(* PLC project PlainProject, Unknown Unnamed 1 *)
(* stored: creationDateTime 2023-09-14T08:06:45, modificationDateTime 2023-09-14T08:09:26 *)

PROGRAM program0
  VAR
    inlet AT %MW0.0.0.20 : INT;
    outlet AT %MW0.0.0.21 : INT;
    level AT %MW0.0.1.0 : INT;
    statustank AT %MW0.0.2.0 : INT;
  END_VAR
  VAR
    pv : INT;
    sp : INT;
    state : INT;
    Setpoint : INT;
    ValveButtonBoth : BOOL;
    tankstatus : INT;
  END_VAR

            pv := level;
sp := Setpoint;
tankstatus := statustank; (* 1=OK, 2=WARNING, 3=BROKEN *)

if ValveButtonBoth then 
state := 4;
else
if pv >= 90 then
state := 1; (* 0= HOLD,  1= DUMP (to not anger management), 2= DRAIN, 3:= FILL *) 
elsif pv > sp + 3 then
state := 2;
elsif pv < sp - 3 then
state :=3;
else
state :=0;
end_if;
end_if;

CASE state OF 
1: inlet := 0;
   outlet := 99;
2: inlet :=0;
   outlet := 70;
3: inlet :=50;
   outlet:=0;
4: inlet :=100;
   outlet :=100; (* expect for the increase due to the tank behaviour *)
0: inlet :=0;
   outlet :=10; (* minimum amount of flow at all times*)
end_case; 













          
END_PROGRAM

CONFIGURATION config
  RESOURCE resource1 ON PLC
    TASK task0(INTERVAL := T#20ms, PRIORITY := 0);
    PROGRAM instance0 WITH task0 : program0;
  END_RESOURCE
END_CONFIGURATION
